RoboDK station: Лабораторная_12.rdk

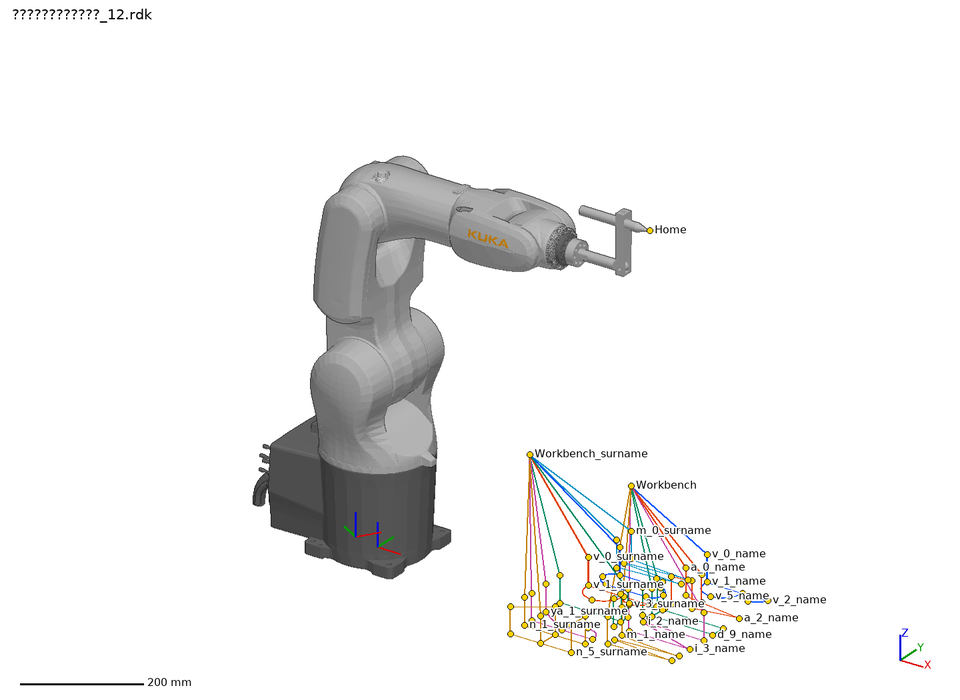
[picture v0: the station drawn from its stored meshes, robots at their saved joint values, targets as dots, program paths as lines]
Station Лабораторная 12 (saved by RoboDK 5.2.5). Poses are relative to the parent item; angles as X-Y-Z fixed-axis rotations.
  - frame KUKA KR 4 R600 Base at (0, 0, 0) mm
    - robot KUKA KR 4 R600: 6 axes, payload 4.63 kg, reach 601 mm, repeatability 0.015 mm, weight 24 kg
        modified DH rows (alpha deg, a mm, theta deg, d mm): 0, 0, 0, 330; -90, 0, 0, 0; 0, 290, -90, 0; -90, 20, 0, 310; 90, 0, 0, 0; -90, 0, 180, 75
        joint limits [-170, -195, -115, -185, -120, -350] to [170, 40, 150, 180, 120, 350]; home [0, -90, 90, 0, 0, 0]; saved at [0, -90, 90, 0, 0, 0]
      - tool , TCP at (-80, 0, 152) mm, rotated rx 180 ry 0 rz 180 deg, size 121.5 x 44 x 157.7 mm
    - target Home (Cartesian target) at (537, 0, 720) mm, rotated rx 0 ry -90 rz 0 deg; joints [0, -90, 90, 0, 0, 0] of KUKA KR 4 R600
    - frame Frame1 at (0, 0, 0) mm
      - target Workbench (Cartesian target) at (500, 0, 250) mm; joints [-24.944, -32.551, 78.534, 0, 44.017, -24.944] of KUKA KR 4 R600
      - target Workbench_surname (Cartesian target) at (300, 0, 250) mm; joints [-24.944, -32.551, 78.534, 0, 44.017, -24.944] of KUKA KR 4 R600
      - target v_0_name (Cartesian target) at (510, 200, 50) mm; joints [-24.944, -32.551, 78.534, 0, 44.017, -24.944] of KUKA KR 4 R600
      - target v_1_name (Cartesian target) at (510, 200, 0) mm; joints [-24.944, -32.551, 78.534, 0, 44.017, -24.944] of KUKA KR 4 R600
      - target v_2_name (Cartesian target) at (630, 200, 0) mm; joints [-24.944, -32.551, 78.534, 0, 44.017, -24.944] of KUKA KR 4 R600
      - target v_3_name (Cartesian target) at (605, 180, 0) mm; joints [-24.944, -32.551, 78.534, 0, 44.017, -24.944] of KUKA KR 4 R600
      - target v_4_name (Cartesian target) at (580, 200, 0) mm; joints [-24.944, -32.551, 78.534, 0, 44.017, -24.944] of KUKA KR 4 R600
      - target v_5_name (Cartesian target) at (545, 160, 0) mm; joints [-24.944, -32.551, 78.534, 0, 44.017, -24.944] of KUKA KR 4 R600
      - target v_0_surname (Cartesian target) at (360, 80, 50) mm; joints [-24.944, -32.551, 78.534, 0, 44.017, -24.944] of KUKA KR 4 R600
      - target v_1_surname (Cartesian target) at (360, 80, 0) mm; joints [-24.944, -32.551, 78.534, 0, 44.017, -24.944] of KUKA KR 4 R600
      - target v_2_surname (Cartesian target) at (480, 80, 0) mm; joints [-24.944, -32.551, 78.534, 0, 44.017, -24.944] of KUKA KR 4 R600
      - target v_3_surname (Cartesian target) at (455, 60, 0) mm; joints [-24.944, -32.551, 78.534, 0, 44.017, -24.944] of KUKA KR 4 R600
      - target v_4_surname (Cartesian target) at (430, 80, 0) mm; joints [-24.944, -32.551, 78.534, 0, 44.017, -24.944] of KUKA KR 4 R600
      - target v_5_surname (Cartesian target) at (395, 40, 0) mm; joints [-24.944, -32.551, 78.534, 0, 44.017, -24.944] of KUKA KR 4 R600
      - target a_0_name (Cartesian target) at (510, 140, 50) mm; joints [-24.944, -32.551, 78.534, 0, 44.017, -24.944] of KUKA KR 4 R600
      - target a_1_name (Cartesian target) at (510, 140, 0) mm; joints [-24.944, -32.551, 78.534, 0, 44.017, -24.944] of KUKA KR 4 R600
      - target a_2_name (Cartesian target) at (630, 120, 0) mm; joints [-24.944, -32.551, 78.534, 0, 44.017, -24.944] of KUKA KR 4 R600
      - target a_3_name (Cartesian target) at (510, 100, 0) mm; joints [-24.944, -32.551, 78.534, 0, 44.017, -24.944] of KUKA KR 4 R600
      - target a_4_name (Cartesian target) at (510, 100, 50) mm; joints [-24.944, -32.551, 78.534, 0, 44.017, -24.944] of KUKA KR 4 R600
      - target a_5_name (Cartesian target) at (546, 106, 50) mm; joints [-24.944, -32.551, 78.534, 0, 44.017, -24.944] of KUKA KR 4 R600
      - target a_6_name (Cartesian target) at (546, 106, 0) mm; joints [-24.944, -32.551, 78.534, 0, 44.017, -24.944] of KUKA KR 4 R600
      - target a_7_name (Cartesian target) at (546, 134, 0) mm; joints [-24.944, -32.551, 78.534, 0, 44.017, -24.944] of KUKA KR 4 R600
      - target a_8_name (Cartesian target) at (546, 134, 50) mm; joints [-24.944, -32.551, 78.534, 0, 44.017, -24.944] of KUKA KR 4 R600
      - target d_0_name (Cartesian target) at (495, 80, 50) mm; joints [-24.944, -32.551, 78.534, 0, 44.017, -24.944] of KUKA KR 4 R600
      - target d_1_name (Cartesian target) at (495, 80, 0) mm; joints [-24.944, -32.551, 78.534, 0, 44.017, -24.944] of KUKA KR 4 R600
      - target d_2_name (Cartesian target) at (510, 80, 0) mm; joints [-24.944, -32.551, 78.534, 0, 44.017, -24.944] of KUKA KR 4 R600
      - target d_3_name (Cartesian target) at (510, 40, 0) mm; joints [-24.944, -32.551, 78.534, 0, 44.017, -24.944] of KUKA KR 4 R600
      - target d_4_name (Cartesian target) at (495, 40, 0) mm; joints [-24.944, -32.551, 78.534, 0, 44.017, -24.944] of KUKA KR 4 R600
      - target d_5_name (Cartesian target) at (495, 40, 50) mm; joints [-24.944, -32.551, 78.534, 0, 44.017, -24.944] of KUKA KR 4 R600
      - target d_6_name (Cartesian target) at (510, 75, 50) mm; joints [-24.944, -32.551, 78.534, 0, 44.017, -24.944] of KUKA KR 4 R600
      - target d_7_name (Cartesian target) at (510, 75, 0) mm; joints [-24.944, -32.551, 78.534, 0, 44.017, -24.944] of KUKA KR 4 R600
      - target d_8_name (Cartesian target) at (630, 75, 0) mm; joints [-24.944, -32.551, 78.534, 0, 44.017, -24.944] of KUKA KR 4 R600
      - target d_9_name (Cartesian target) at (630, 45, 0) mm; joints [-24.944, -32.551, 78.534, 0, 44.017, -24.944] of KUKA KR 4 R600
      - target d_10_name (Cartesian target) at (510, 45, 0) mm; joints [-24.944, -32.551, 78.534, 0, 44.017, -24.944] of KUKA KR 4 R600
      - target d_11_name (Cartesian target) at (510, 45, 50) mm; joints [-24.944, -32.551, 78.534, 0, 44.017, -24.944] of KUKA KR 4 R600
      - target i_0_name (Cartesian target) at (630, 20, 50) mm; joints [-24.944, -32.551, 78.534, 0, 44.017, -24.944] of KUKA KR 4 R600
      - target i_1_name (Cartesian target) at (630, 20, 0) mm; joints [-24.944, -32.551, 78.534, 0, 44.017, -24.944] of KUKA KR 4 R600
      - target i_2_name (Cartesian target) at (510, 20, 0) mm; joints [-24.944, -32.551, 78.534, 0, 44.017, -24.944] of KUKA KR 4 R600
      - target i_3_name (Cartesian target) at (630, -20, 0) mm; joints [-24.944, -32.551, 78.534, 0, 44.017, -24.944] of KUKA KR 4 R600
      - target i_4_name (Cartesian target) at (510, -20, 0) mm; joints [-24.944, -32.551, 78.534, 0, 44.017, -24.944] of KUKA KR 4 R600
      - target i_5_name (Cartesian target) at (510, -20, 50) mm; joints [-24.944, -32.551, 78.534, 0, 44.017, -24.944] of KUKA KR 4 R600
      - target m_0_name (Cartesian target) at (510, -40, 50) mm; joints [-24.944, -32.551, 78.534, 0, 44.017, -24.944] of KUKA KR 4 R600
      - target m_1_name (Cartesian target) at (510, -40, 0) mm; joints [-24.944, -32.551, 78.534, 0, 44.017, -24.944] of KUKA KR 4 R600
      - target m_2_name (Cartesian target) at (630, -50, 0) mm; joints [-24.944, -32.551, 78.534, 0, 44.017, -24.944] of KUKA KR 4 R600
      - target m_3_name (Cartesian target) at (510, -60, 0) mm; joints [-24.944, -32.551, 78.534, 0, 44.017, -24.944] of KUKA KR 4 R600
      - target m_4_name (Cartesian target) at (630, -70, 0) mm; joints [-24.944, -32.551, 78.534, 0, 44.017, -24.944] of KUKA KR 4 R600
      - target m_5_name (Cartesian target) at (510, -80, 0) mm; joints [-24.944, -32.551, 78.534, 0, 44.017, -24.944] of KUKA KR 4 R600
      - target m_6_name (Cartesian target) at (510, -80, 50) mm; joints [-24.944, -32.551, 78.534, 0, 44.017, -24.944] of KUKA KR 4 R600
      - target m_0_surname (Cartesian target) at (360, 200, 50) mm; joints [-24.944, -32.551, 78.534, 0, 44.017, -24.944] of KUKA KR 4 R600
      - target m_1_surname (Cartesian target) at (360, 200, 0) mm; joints [-24.944, -32.551, 78.534, 0, 44.017, -24.944] of KUKA KR 4 R600
      - target m_2_surname (Cartesian target) at (480, 190, 0) mm; joints [-24.944, -32.551, 78.534, 0, 44.017, -24.944] of KUKA KR 4 R600
      - target m_3_surname (Cartesian target) at (360, 180, 0) mm; joints [-24.944, -32.551, 78.534, 0, 44.017, -24.944] of KUKA KR 4 R600
      - target m_4_surname (Cartesian target) at (480, 170, 0) mm; joints [-24.944, -32.551, 78.534, 0, 44.017, -24.944] of KUKA KR 4 R600
      - target m_5_surname (Cartesian target) at (360, 160, 0) mm; joints [-24.944, -32.551, 78.534, 0, 44.017, -24.944] of KUKA KR 4 R600
      - target m_6_surname (Cartesian target) at (360, 160, 50) mm; joints [-24.944, -32.551, 78.534, 0, 44.017, -24.944] of KUKA KR 4 R600
      - target o_0_surname (Cartesian target) at (380, 140, 50) mm; joints [-24.944, -32.551, 78.534, 0, 44.017, -24.944] of KUKA KR 4 R600
      - target o_1_surname (Cartesian target) at (380, 140, 0) mm; joints [-24.944, -32.551, 78.534, 0, 44.017, -24.944] of KUKA KR 4 R600
      - target o_2_surname (Cartesian target) at (360, 120, 0) mm; joints [-24.944, -32.551, 78.534, 0, 44.017, -24.944] of KUKA KR 4 R600
      - target o_3_surname (Cartesian target) at (380, 100, 0) mm; joints [-24.944, -32.551, 78.534, 0, 44.017, -24.944] of KUKA KR 4 R600
      - target o_4_surname (Cartesian target) at (460, 100, 0) mm; joints [-24.944, -32.551, 78.534, 0, 44.017, -24.944] of KUKA KR 4 R600
      - target o_5_surname (Cartesian target) at (480, 120, 0) mm; joints [-24.944, -32.551, 78.534, 0, 44.017, -24.944] of KUKA KR 4 R600
      - target o_6_surname (Cartesian target) at (460, 140, 0) mm; joints [-24.944, -32.551, 78.534, 0, 44.017, -24.944] of KUKA KR 4 R600
      - target t_0_surname (Cartesian target) at (480, 20, 50) mm; joints [-24.944, -32.551, 78.534, 0, 44.017, -24.944] of KUKA KR 4 R600
      - target t_1_surname (Cartesian target) at (480, 20, 0) mm; joints [-24.944, -32.551, 78.534, 0, 44.017, -24.944] of KUKA KR 4 R600
      - target t_2_surname (Cartesian target) at (480, -20, 0) mm; joints [-24.944, -32.551, 78.534, 0, 44.017, -24.944] of KUKA KR 4 R600
      - target t_3_surname (Cartesian target) at (480, -20, 50) mm; joints [-24.944, -32.551, 78.534, 0, 44.017, -24.944] of KUKA KR 4 R600
      - target t_4_surname (Cartesian target) at (480, 0, 50) mm; joints [-24.944, -32.551, 78.534, 0, 44.017, -24.944] of KUKA KR 4 R600
      - target t_5_surname (Cartesian target) at (480, 0, 0) mm; joints [-24.944, -32.551, 78.534, 0, 44.017, -24.944] of KUKA KR 4 R600
      - target t_6_surname (Cartesian target) at (360, 0, 0) mm; joints [-24.944, -32.551, 78.534, 0, 44.017, -24.944] of KUKA KR 4 R600
      - target t_7_surname (Cartesian target) at (360, 0, 50) mm; joints [-24.944, -32.551, 78.534, 0, 44.017, -24.944] of KUKA KR 4 R600
      - target ya_0_surname (Cartesian target) at (360, -40, 50) mm; joints [-24.944, -32.551, 78.534, 0, 44.017, -24.944] of KUKA KR 4 R600
      - target ya_1_surname (Cartesian target) at (360, -40, 0) mm; joints [-24.944, -32.551, 78.534, 0, 44.017, -24.944] of KUKA KR 4 R600
      - target ya_2_surname (Cartesian target) at (420, -80, 0) mm; joints [-24.944, -32.551, 78.534, 0, 44.017, -24.944] of KUKA KR 4 R600
      - target ya_3_surname (Cartesian target) at (450, -50, 0) mm; joints [-24.944, -32.551, 78.534, 0, 44.017, -24.944] of KUKA KR 4 R600
      - target ya_4_surname (Cartesian target) at (480, -80, 0) mm; joints [-24.944, -32.551, 78.534, 0, 44.017, -24.944] of KUKA KR 4 R600
      - target ya_5_surname (Cartesian target) at (360, -80, 0) mm; joints [-24.944, -32.551, 78.534, 0, 44.017, -24.944] of KUKA KR 4 R600
      - target ya_6_surname (Cartesian target) at (360, -80, 50) mm; joints [-24.944, -32.551, 78.534, 0, 44.017, -24.944] of KUKA KR 4 R600
      - target n_0_surname (Cartesian target) at (360, -100, 50) mm; joints [-24.944, -32.551, 78.534, 0, 44.017, -24.944] of KUKA KR 4 R600
      - target n_1_surname (Cartesian target) at (360, -100, 0) mm; joints [-24.944, -32.551, 78.534, 0, 44.017, -24.944] of KUKA KR 4 R600
      - target n_2_surname (Cartesian target) at (480, -100, 0) mm; joints [-24.944, -32.551, 78.534, 0, 44.017, -24.944] of KUKA KR 4 R600
      - target n_3_surname (Cartesian target) at (480, -100, 50) mm; joints [-24.944, -32.551, 78.534, 0, 44.017, -24.944] of KUKA KR 4 R600
      - target n_4_surname (Cartesian target) at (480, -140, 50) mm; joints [-24.944, -32.551, 78.534, 0, 44.017, -24.944] of KUKA KR 4 R600
      - target n_5_surname (Cartesian target) at (480, -140, 0) mm; joints [-24.944, -32.551, 78.534, 0, 44.017, -24.944] of KUKA KR 4 R600
      - target n_6_surname (Cartesian target) at (360, -140, 0) mm; joints [-24.944, -32.551, 78.534, 0, 44.017, -24.944] of KUKA KR 4 R600
      - target n_7_surname (Cartesian target) at (360, -140, 50) mm; joints [-24.944, -32.551, 78.534, 0, 44.017, -24.944] of KUKA KR 4 R600
      - target n_8_surname (Cartesian target) at (420, -100, 50) mm; joints [-24.944, -32.551, 78.534, 0, 44.017, -24.944] of KUKA KR 4 R600
      - target n_9_surname (Cartesian target) at (420, -100, 0) mm; joints [-24.944, -32.551, 78.534, 0, 44.017, -24.944] of KUKA KR 4 R600
      - target n_10_surname (Cartesian target) at (420, -140, 0) mm; joints [-24.944, -32.551, 78.534, 0, 44.017, -24.944] of KUKA KR 4 R600
      - target n_11_surname (Cartesian target) at (420, -140, 50) mm; joints [-24.944, -32.551, 78.534, 0, 44.017, -24.944] of KUKA KR 4 R600
    - frame Frame_turned at (-50, 10, 0) mm, rotated rx 0 ry 0 rz 60 deg
  - program Full (2 instructions, listed below)
  - program letter_v (13 instructions, listed below)
  - program letter_a (18 instructions, listed below)
  - program letter_d (21 instructions, listed below)
  - program letter_i (13 instructions, listed below)
  - program letter_m (14 instructions, listed below)
  - program letter_m_surname (14 instructions, listed below)
  - program letter_o_surname (14 instructions, listed below)
  - program letter_v_surname (13 instructions, listed below)
  - program letter_t_surname (17 instructions, listed below)
  - program letter_ya_surname (13 instructions, listed below)
  - program letter_n_surname (23 instructions, listed below)
  - program Main (16 instructions, listed below)
  - program Rotate (16 instructions, listed below)
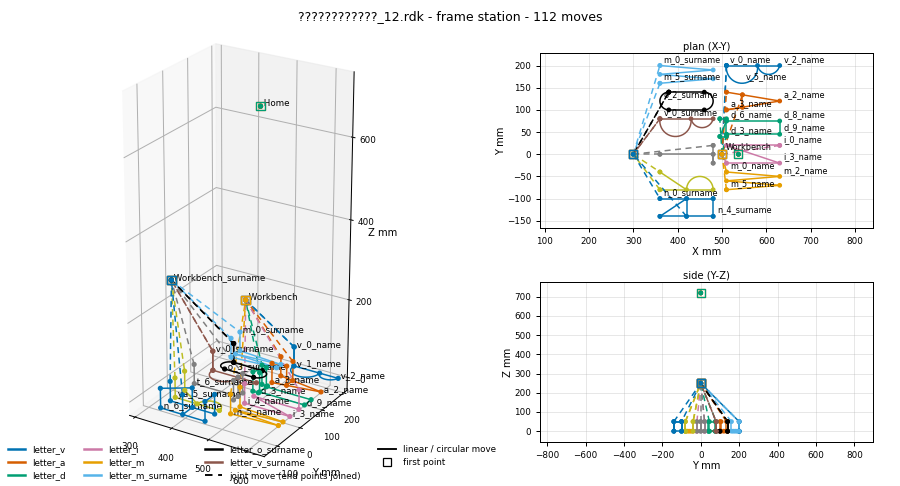
[picture p0: tool path of Лабораторная_12.rdk in frame station, 112 of 112 moves have a stored position in this frame; points joined in program order, loops and branches not executed]

--- program Full (robot KUKA KR 4 R600) ---
  Call Main
  Call Rotate

--- program letter_v (robot KUKA KR 4 R600) ---
  Set speed (100.0 mm/s)
  MoveJ (Workbench)
  MoveJ (v_0_name)
  Set speed (50.0 mm/s)
  MoveL (v_1_name)
  Set speed (75.0 mm/s)
  MoveL (v_2_name)
  MoveC (v_3_name, v_4_name)
  MoveC (v_5_name, v_1_name)
  Set speed (50.0 mm/s)
  MoveL (v_0_name)
  Set speed (100.0 mm/s)
  MoveJ (Workbench)

--- program letter_a (robot KUKA KR 4 R600) ---
  Set speed (100.0 mm/s)
  MoveJ (Workbench)
  MoveJ (a_0_name)
  Set speed (50.0 mm/s)
  MoveL (a_1_name)
  Set speed (75.0 mm/s)
  MoveL (a_2_name)
  MoveL (a_3_name)
  Set speed (50.0 mm/s)
  MoveL (a_4_name)
  MoveL (a_5_name)
  MoveL (a_6_name)
  Set speed (75.0 mm/s)
  MoveL (a_7_name)
  Set speed (50.0 mm/s)
  MoveL (a_8_name)
  Set speed (100.0 mm/s)
  MoveJ (Workbench)

--- program letter_d (robot KUKA KR 4 R600) ---
  Set speed (100.0 mm/s)
  MoveJ (Workbench)
  MoveJ (d_0_name)
  Set speed (50.0 mm/s)
  MoveL (d_1_name)
  Set speed (75.0 mm/s)
  MoveL (d_2_name)
  MoveL (d_3_name)
  MoveL (d_4_name)
  Set speed (50.0 mm/s)
  MoveL (d_5_name)
  MoveL (d_6_name)
  MoveL (d_7_name)
  Set speed (75.0 mm/s)
  MoveL (d_8_name)
  MoveL (d_9_name)
  MoveL (d_10_name)
  Set speed (50.0 mm/s)
  MoveL (d_11_name)
  Set speed (100.0 mm/s)
  MoveJ (Workbench)

--- program letter_i (robot KUKA KR 4 R600) ---
  Set speed (100.0 mm/s)
  MoveJ (Workbench)
  MoveJ (i_0_name)
  Set speed (50.0 mm/s)
  MoveL (i_1_name)
  Set speed (75.0 mm/s)
  MoveL (i_2_name)
  MoveL (i_3_name)
  MoveL (i_4_name)
  Set speed (50.0 mm/s)
  MoveL (i_5_name)
  Set speed (100.0 mm/s)
  MoveJ (Workbench)

--- program letter_m (robot KUKA KR 4 R600) ---
  Set speed (100.0 mm/s)
  MoveJ (Workbench)
  MoveJ (m_0_name)
  Set speed (50.0 mm/s)
  MoveL (m_1_name)
  Set speed (75.0 mm/s)
  MoveL (m_2_name)
  MoveL (m_3_name)
  MoveL (m_4_name)
  MoveL (m_5_name)
  Set speed (50.0 mm/s)
  MoveL (m_6_name)
  Set speed (100.0 mm/s)
  MoveJ (Workbench)

--- program letter_m_surname (robot KUKA KR 4 R600) ---
  Set speed (100.0 mm/s)
  MoveJ (Workbench_surname)
  MoveJ (m_0_surname)
  Set speed (50.0 mm/s)
  MoveL (m_1_surname)
  Set speed (75.0 mm/s)
  MoveL (m_2_surname)
  MoveL (m_3_surname)
  MoveL (m_4_surname)
  MoveL (m_5_surname)
  Set speed (50.0 mm/s)
  MoveL (m_6_surname)
  Set speed (100.0 mm/s)
  MoveJ (Workbench_surname)

--- program letter_o_surname (robot KUKA KR 4 R600) ---
  Set speed (100.0 mm/s)
  MoveJ (Workbench_surname)
  MoveJ (o_0_surname)
  Set speed (50.0 mm/s)
  MoveL (o_1_surname)
  Set speed (75.0 mm/s)
  MoveC (o_2_surname, o_3_surname)
  MoveL (o_4_surname)
  MoveC (o_5_surname, o_6_surname)
  MoveL (o_1_surname)
  Set speed (50.0 mm/s)
  MoveL (o_0_surname)
  Set speed (100.0 mm/s)
  MoveJ (Workbench_surname)

--- program letter_v_surname (robot KUKA KR 4 R600) ---
  Set speed (100.0 mm/s)
  MoveJ (Workbench_surname)
  MoveJ (v_0_surname)
  Set speed (50.0 mm/s)
  MoveL (v_1_surname)
  Set speed (75.0 mm/s)
  MoveL (v_2_surname)
  MoveC (v_3_surname, v_4_surname)
  MoveC (v_5_surname, v_1_surname)
  Set speed (50.0 mm/s)
  MoveL (v_0_surname)
  Set speed (100.0 mm/s)
  MoveJ (Workbench_surname)

--- program letter_t_surname (robot KUKA KR 4 R600) ---
  Set speed (100.0 mm/s)
  MoveJ (Workbench_surname)
  MoveJ (t_0_surname)
  Set speed (50.0 mm/s)
  MoveL (t_1_surname)
  Set speed (75.0 mm/s)
  MoveL (t_2_surname)
  Set speed (50.0 mm/s)
  MoveL (t_3_surname)
  MoveL (t_4_surname)
  MoveL (t_5_surname)
  Set speed (75.0 mm/s)
  MoveL (t_6_surname)
  Set speed (50.0 mm/s)
  MoveL (t_7_surname)
  Set speed (100.0 mm/s)
  MoveJ (Workbench_surname)

--- program letter_ya_surname (robot KUKA KR 4 R600) ---
  Set speed (100.0 mm/s)
  MoveJ (Workbench_surname)
  MoveJ (ya_0_surname)
  Set speed (50.0 mm/s)
  MoveL (ya_1_surname)
  Set speed (75.0 mm/s)
  MoveL (ya_2_surname)
  MoveC (ya_3_surname, ya_4_surname)
  MoveL (ya_5_surname)
  Set speed (50.0 mm/s)
  MoveL (ya_6_surname)
  Set speed (100.0 mm/s)
  MoveJ (Workbench_surname)

--- program letter_n_surname (robot KUKA KR 4 R600) ---
  Set speed (100.0 mm/s)
  MoveJ (Workbench_surname)
  MoveJ (n_0_surname)
  Set speed (50.0 mm/s)
  MoveL (n_1_surname)
  Set speed (75.0 mm/s)
  MoveL (n_2_surname)
  Set speed (50.0 mm/s)
  MoveL (n_3_surname)
  MoveL (n_4_surname)
  MoveL (n_5_surname)
  Set speed (75.0 mm/s)
  MoveL (n_6_surname)
  Set speed (50.0 mm/s)
  MoveL (n_7_surname)
  MoveL (n_8_surname)
  MoveL (n_9_surname)
  Set speed (75.0 mm/s)
  MoveL (n_10_surname)
  Set speed (50.0 mm/s)
  MoveL (n_11_surname)
  Set speed (100.0 mm/s)
  MoveJ (Workbench_surname)

--- program Main (robot KUKA KR 4 R600) ---
  Set Ref.: KUKA KR 4 R600 Base
  MoveJ (Home)
  Set Ref.: Frame1
  Call letter_v
  Call letter_a
  Call letter_d
  Call letter_i
  Call letter_m
  Call letter_m_surname
  Call letter_o_surname
  Call letter_v_surname
  Call letter_t_surname
  Call letter_ya_surname
  Call letter_n_surname
  Set Ref.: KUKA KR 4 R600 Base
  MoveJ (Home)

--- program Rotate (robot KUKA KR 4 R600) ---
  Set Ref.: KUKA KR 4 R600 Base
  MoveJ (Home)
  Set Ref.: Frame_turned
  Call letter_v
  Call letter_a
  Call letter_d
  Call letter_i
  Call letter_m
  Call letter_m_surname
  Call letter_o_surname
  Call letter_v_surname
  Call letter_t_surname
  Call letter_ya_surname
  Call letter_n_surname
  Set Ref.: KUKA KR 4 R600 Base
  MoveJ (Home)
